(* Logix 5000 project; controller PBS_Perfusion vendor 1 type 14 code 217 rev 32.14; software revision 32.03; part 14 of 27 *)
(* tags used below, declared in another part *)
   Inp_OnFdbk : BOOL;   // Input Signal: ON feedback from device
   Inp_OffFdbk : BOOL;   // Input Signal: OFF feedback from device
   Inp_PermOK : BOOL;   // 1=ON Permissives OK, device can turn ON
   Inp_NBPermOK : BOOL;   // 1=Non-Bypassable ON Permissives OK, device can turn ON
   Inp_IntlkOK : BOOL;   // 1=Interlocks OK, device can turn ON and stay ON
   Inp_NBIntlkOK : BOOL;   // 1=Non-Bypassable Interlocks OK, device can turn ON and stay ON
   Inp_IntlkAvail : BOOL;   // 1 = Interlock Availibility OK
   Inp_IOFault : BOOL;   // Input Communication Status 0=OK, 1=fail
   Inp_Sim : BOOL;   // 1=Simulate working device; 0=Turn ON/OFF actual device
   Inp_OvrdCmd : DINT;   // Ovrd Device Command 0=None, 1=Off, 2=On, 3=Pulse Off, 4=Pulse On, 5=Pulse Cont
   Inp_HornInh : BOOL;   // 1 = Inhibit audible alert, 0 = Alllow audible alert
   Inp_Reset : BOOL;   // 1=Reset Shed Latches and Cleared Alarms
   Cfg_HasPulse : BOOL;   // 1=Enable pulsing functions, 0=On/Off only
   Cfg_HasOnFdbk : BOOL;   // 1=Device provides an ON feedback signal
   Cfg_HasOffFdbk : BOOL;   // 1=Device provides an OFF feedback signal
   Cfg_UseOnFdbk : BOOL;   // 1=Device ON feedback should be used for failure checking
   Cfg_UseOffFdbk : BOOL;   // 1=Device OFF feedback should be used for failure checking
   Cfg_FdbkFail : BOOL;   // 1=Both feedbacks ON is invalid; 0=Both feedbacks OFF is invalid
   Cfg_HasMoreObj : BOOL;   // 1=Tells HMI an object with more info is available
   Cfg_HornOnChange : BOOL;   // 0 = Horn on energize only, 1 = Horn on any state change
   Cfg_OperOffPrio : BOOL;   // 1=OCmd_Off any time, 0=OCmd_Off only when Oper selected
   Cfg_ExtOffPrio : BOOL;   // 1=XCmd_Off any time, 0=XCmd_Off only when Oper selected
   Cfg_OCmdResets : BOOL;   // 1=New device OCmd resets shed latches and cleared alarms, 0=OCmdReset req'd.
   Cfg_XCmdResets : BOOL;   // 1=New device XCmd resets shed latches and cleared alarms, 0=XCmdReset req'd.
   Cfg_OvrdPermIntlk : BOOL;   // 1=Override ignores Bypassable Perm/ Intlk; 0=always use Perm/Intlk
   Cfg_ShedOnFail : BOOL;   // 1=Go to State 0 and Alarm on Fail to reach position; 0=Alarm only on Fail
   Cfg_ShedOnIOFault : BOOL;   // 1=Go to State 0 and Alarm on I/O Fault; 0=Alarm only on I/O Fault
   Cfg_StartHornT : REAL;   // Time to sound audible on commanded start (sec) (0=disabled)
   Cfg_SimFdbkT : REAL;   // Delay to echo back of ON/OFF status when in Simulation (sec)
   Cfg_OnDelayT : REAL;   // Delay before initially turning output ON (sec)
   Cfg_OffDelayT : REAL;   // Delay before initially turning output OFF (sec)
   Cfg_OnPulseT : REAL;   // Output ON time for Pulse ON or Pulse Continuous
   Cfg_OffPulseT : REAL;   // Output OFF time for Pulse OFF or Pulse Continuous
   Cfg_OnFailT : REAL;   // Time after Output ON to get ON Feedback before Fault (sec)
   Cfg_OffFailT : REAL;   // Time after Output OFF to get OFF Feedback before Fault (sec)
   PSet_Owner : DINT;   // Program Owner Request ID (non-zero) or Release (zero)
   PCmd_On : BOOL;   // Program Command to turn device ON
   PCmd_Off : BOOL;   // Program Command to turn device OFF
   PCmd_OnPulse : BOOL;   // Program Command to pulse device (which is OFF) ON once
   PCmd_OffPulse : BOOL;   // Program Command to pulse device (which is ON) OFF once
   PCmd_ContPulse : BOOL;   // Program Command to pulse device continuously (blink)
   PCmd_Reset : BOOL;   // Program Command to ResetShed Latches and Cleared Alarms
   PCmd_OnFailAck : ALIAS FOR OnFail.PCmd_Ack;   // Program Command to Acknowledge Fail to Turn ON Alarm
   PCmd_OffFailAck : ALIAS FOR OffFail.PCmd_Ack;   // Program Command to Acknowledge Fail to Turn OFF Alarm
   PCmd_IntlkTripAck : ALIAS FOR IntlkTrip.PCmd_Ack;   // Program Command to Acknowledge Interlock Trip Alarm
   PCmd_IOFaultAck : ALIAS FOR IOFault.PCmd_Ack;   // Program Command to Acknowledge I/O Fault Alarm
   XCmd_On : BOOL;   // External Command to turn device ON
   XCmd_Off : BOOL;   // External Command to turn device OFF
   XCmd_OnPulse : BOOL;   // External Command to pulse device (which is OFF) ON once
   XCmd_OffPulse : BOOL;   // External Command to pulse device (which is ON) OFF once
   XCmd_ContPulse : BOOL;   // External Command to pulse device continuously (blink)
   XCmd_Reset : BOOL;   // Ext Cmd to clear shed latches and cleared alarms
   Out : BOOL;   // Primary Output 1=ON, 0=OFF
   Val_Fdbk : DINT;   // Device Feedback: 0=Transition, 1=Off, 2=On, 3=Invalid
   Val_Sts : DINT;   // Device Status 0=off 1=on 2=pulse off 3=pulse on 4=pulse cont. 5=turning off 6=turning on
   Val_Owner : DINT;   // Current Object Owner ID (0=not owned)
   Sts_FdbkOff : BOOL;   // 1=Device Feedback shows device in OFF state
   Sts_FdbkOn : BOOL;   // 1=Device Feedback shows device in ON state
   Sts_FdbkFail : BOOL;   // 1=Feedbacks are in an INVALID state (not ON, OFF or TRANSIT)
   Sts_Available : BOOL;   // 1=Device available for control by automation (Prog)
   Sts_Bypass : BOOL;   // 1=Bypassable Interlocks and Permissives are Bypassed
   Sts_BypActive : BOOL;   // 1=Interlock / Permissive Bypassing Active (Bypassed or Maintenance)
   Sts_NotRdy : BOOL;   // 1=Device Not Ready, see detail bits for reason
   Nrdy_CfgErr : BOOL;   // 1=Device Not Ready: Configuration Error
   Nrdy_Fail : BOOL;   // 1=Device Not Ready: Device Failure (Shed Requires Reset)
   Nrdy_Intlk : BOOL;   // 1=Device Not Ready: Interlock Not OK
   Nrdy_IOFault : BOOL;   // 1=Device Not Ready: I/O Fault (Shed Requires Reset)
   Nrdy_OoS : BOOL;   // 1=Device Not Ready: Device is Out of Service
   Nrdy_PrioOff : BOOL;   // 1=Device Not Ready: Oper/Ext Priority Off Comand Requires Reset
   Nrdy_Perm : BOOL;   // 1=Device Not Ready: Permissive Not OK
   Sts_MaintByp : BOOL;   // 1=Device has a Maintenance Bypass function active
   Err_Timer : BOOL;   // 1=Error in Config: Feeback Check timer preset (use 0 to 2147483)
   Err_Sim : BOOL;   // 1=Error in Config: Simulation timer preset (use 0 to 2147483)
   Sts_Hand : ALIAS FOR CmdSrc.Sts_Hand;
   Sts_OoS : ALIAS FOR CmdSrc.Sts_OoS;
   Sts_Maint : ALIAS FOR CmdSrc.Sts_Maint;
   Sts_Ovrd : ALIAS FOR CmdSrc.Sts_Ovrd;
   Sts_Ext : ALIAS FOR CmdSrc.Sts_Ext;
   Sts_Prog : ALIAS FOR CmdSrc.Sts_Prog;
   Sts_Oper : ALIAS FOR CmdSrc.Sts_Oper;
   Sts_OnFail : ALIAS FOR OnFail.Inp;   // 1=Device Failed to Turn ON
   Sts_OffFail : ALIAS FOR OffFail.Inp;   // 1=Device Failed to Turn OFF
   Sts_IntlkTrip : ALIAS FOR IntlkTrip.Inp;   // 1=Device turned OFF by an Interlock NOT OK (one-shot)
   Sts_IOFault : ALIAS FOR IOFault.Inp;   // I/O Comm Fault Status (0=OK, 1=Bad)
   P_DOut : BOOL;   // Unique Parameter Name for auto - discovery
   Wrk_OffT : TIMER;   // Off Feedback Check Timer
   Wrk_OnT : TIMER;   // On Feedback Check Timer
   Wrk_SimOffT : TIMER;   // Simulation Delay until OFF
   Wrk_SimOnT : TIMER;   // Simulation Delay until ON
   Wrk_OnFdbk : BOOL;   // ON Feedback based on Command Source, simulation, etc. 1=confirmed ON
   Wrk_Bypass : BOOL;   // Internal Bypassable Permissives and Interlocks are Bypassed flag
   CmdSrc : P_CmdSrc;   // Control / Command Source Selection
   IOFault : P_Alarm;   // I/O Fault Alarm
   IntlkTrip : P_Alarm;   // Interlock Trip Alarm
   OffFail : P_Alarm;   // Device Failed to Turn OFF Alarm
   OnFail : P_Alarm;   // Device Failed to Turn ON Alarm
   Cfg_Tag : STRING_20;   // Tagname for display on HMI
   Cfg_Label : STRING_20;   // Label for graphic symbol displayed on HMI
   Cfg_Desc : STRING_40;   // Description for display on HMI
   Wrk_OffFdbk : BOOL;   // OFF Feedback based on Command Source, simulation, etc. 1=confirmed OFF
   Wrk_OnPulseT : TIMER;   // Output ON Pulse Timer
   Wrk_OffPulseT : TIMER;   // Output OFF Pulse Timer
   Wrk_OffDelayT : TIMER;   // Dealy before turning output OFF (Timer)
   Wrk_OnDelayT : TIMER;   // Delay before turning output ON (Timer)
   Wrk_PermOK : BOOL;   // 1=Permissives are all OK to energize
   Wrk_Cmd : DINT;   // Device Command: 0= None, bit .0=Off, bit .1=On, bit .2=Pulse Off, bit .3=Pulse On, bit .4=Pulse Cont.
   Cfg_1StText : STRING_8;   // Text to display in PV=1 State
   Cfg_0StText : STRING_8;   // Text to display in PV=0 State
   HMI_Type : STRING_16;   // Type identifier for HMI navigation
   HMI_Lib : STRING_12;   // Display Library for Faceplate call-up
   Wrk_NotRdy : BOOL;   // Device Not Ready conditions excluding shed latches
   Wrk_NoLongerSim : BOOL;   // Switched from Simulated to Real Device this scan
   Cfg_Area : STRING_Area;   // Process Area for security
   OCmd_ResetAckAll : BOOL;   // Operator Command to Reset all Alarms and latched Shed conditions
   OCmd_Reset : BOOL;   // Operator Command to Reset all Alarms requiring Reset
   OCmd_ContPulse : BOOL;   // Operator Command to pulse device continuously (blink)
   OCmd_OffPulse : BOOL;   // Operator Command to pulse device (which is ON) OFF once
   OCmd_OnPulse : BOOL;   // Operator Command to pulse device (which is OFF) ON once
   OCmd_Off : BOOL;   // Operator Command to turn device OFF
   OCmd_On : BOOL;   // Operator Command to turn device ON
   MCmd_Check : BOOL;   // Maintenance Command to Check (not bypass) all Interlocks and Permissives
   MCmd_Bypass : BOOL;   // Maintenance Command to Bypass all Bypassable Interlocks and Permissives
   MRdy_Check : BOOL;   // 1=Ready for MCmd_Check (enables HMI button)
   MRdy_Bypass : BOOL;   // 1=Ready for MCmd_Bypass (enables HMI button)
   Wrk_State : DINT;   // Internal value of state machine current state
   Wrk_StartHornT : TIMER;   // Timer for audible alert or start
   Wrk_StartHorn : BOOL;   // 1=Sound audible prior to commanded energize/ state change
   ONS : DINT[3];
   REAL : DINT;
(* P_DOut, continued *)

ROUTINE Logic   (* ladder *)
// Control Discrete Output, monitoring Feedbacks
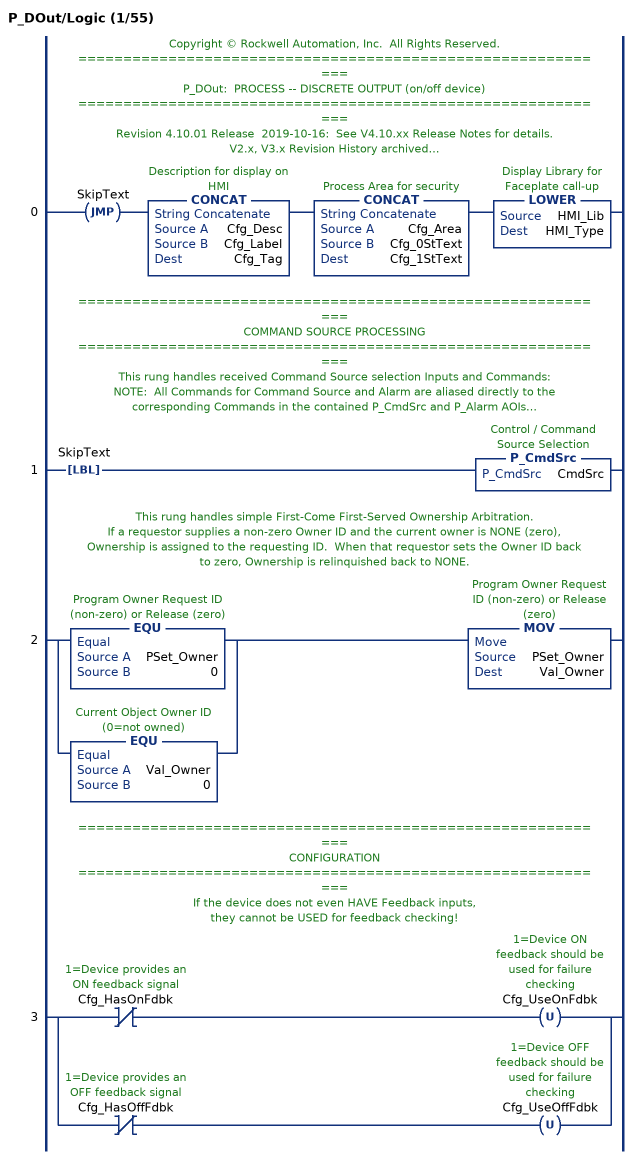
   // Copyright © Rockwell Automation, Inc.  All Rights Reserved.
   // ============================================================
   // P_DOut:  PROCESS -- DISCRETE OUTPUT (on/off device)
   // ============================================================
   // Revision 4.10.01 Release  2019-10-16:  See V4.10.xx Release Notes for details.
   // V2.x, V3.x Revision History archived.
   // V4.00.00  2018-07-02:  Changed "Mode" to "Command Source". Changed Inf_
   // items to HMI_, and added Cfg_Area for security. Added unacked alarm count.
   // Deleted Cfg_PCmdClear; all Program Commands are now self-clearing.
   // Added option: Cfg_HasPulse. Aligned ready bit naming with command bit names.
   // Changed delay / time configuration items to REAL seconds.
   // V4.00.02  2018-10-30:  Fixed feedback determination for simulation or no feedback.
   // V4.10.00  2019-10-16:  Added audible alert on commanded energize/state change.
   // Added Horn Status, Horn Inhibit. Changed availability to use input availability
   // from interlocks. Updated to P_CmdSrc V4.10.00. Added Cfg_HasMoreObj.
   // V4.10.01  2019-10-11:  Corrected operation of state machine with alert horn.
   // ============================================================
   // This Instruction controls (and optionally monitors feedback for)
   // a single Discrete Output and provides:
   // *  Operator and Program Commands to:
   //     -  turn the output ON
   //     -  turn the output OFF
   //     -  if the output is OFF, pulse it ON for a configured time
   //     -  if the output is ON, pulse it OFF for a configured time, or
   //     -  pulse the output continuously at the configured ON
   //         and OFF times (e.g., for blinking a lamp)
   // *  User-configurable ON delay and OFF delay before first output change
   // *  User-configurable text labels for the ON and OFF states
   // *  Optional monitoring of ON and OFF state confirmation feedbacks
   // *  Detection of Failure to turn ON or OFF (when feedbacks are used)
   // *  Monitoring of Permissive conditions to allow energizing output
   // *  Monitoring of Interlock conditions to de-energize output
   // *  Optional return to previous state upon return from Hand,
   //       Override, or Interlock
   // *  Simulation, providing feedback of a working device while
   //       disabling output (keeping de-energized)
   // *  Monitoring of I/O communication faults
   // *  Alarms for Fail to Turn ON, Fail to turn OFF (if feedbacks are
   //       used), Interlock Trip, I/O Fault
   // *  "Available" status for use by automation logic to know whether
   //       output can be controlled by other objects.
   // Command Sources are arbitrated by a P_CmdSrc Add-On Instruction instance.
   // Command Sources: Operator, External, Program, External, Override, Maintenance,
   // Out of Service, Hand.  Alarms are provided by P_Alarm Add-On Instruction instances.
   // ============================================================
   // SHOW LOCAL STRINGS
   // ============================================================
   // The STRINGs containing the text associated with each instance of this
   // instruction cannot be Input or Output Parameters, because STRINGs are not
   //  'atomic' types. (Inputs and Outputs must be SINT, INT, DINT, REAL, or BOOL.)
   // In order to make it easier to find and configure these STRINGs, this rung
   // was added.  THE JMP (and the LBL on the following rung)
   // MUST NOT BE REMOVED!!!
   // To view the STRINGs, go to the instruction instance (in LD or FBD), RIGHT-click
   // to bring up the context menu and select "Open Instruction Logic".
   // This rung will appear with the STRING values for the selected instance.
   // You may double-click the STRING values here to modify them as well.
   // #####  V4.00.00  2018-07-02:  Added string for Cfg_Area, renamed Inf_* to HMI_*.  #####
   0: JMP(SkipText)CONCAT(Cfg_Desc,Cfg_Label,Cfg_Tag)CONCAT(Cfg_Area,Cfg_0StText,Cfg_1StText)LOWER(HMI_Lib,HMI_Type);
   // ============================================================
   // COMMAND SOURCE PROCESSING
   // ============================================================
   // This rung handles received Command Source selection Inputs and Commands:
   // NOTE:  All Commands for Command Source and Alarm are aliased directly to the
   // corresponding Commands in the contained P_CmdSrc and P_Alarm AOIs.
   // #####  V4.00.00  2018-07-02:  Changed P_Mode to P_CmdSrc.  #####
   1: LBL(SkipText)P_CmdSrc(CmdSrc);
   // This rung handles simple First-Come First-Served Ownership Arbitration.
   // If a requestor supplies a non-zero Owner ID and the current owner is NONE (zero),
   // Ownership is assigned to the requesting ID.  When that requestor sets the Owner ID back
   // to zero, Ownership is relinquished back to NONE.
   2: [EQU(PSet_Owner,0) ,EQU(Val_Owner,0) ]MOV(PSet_Owner,Val_Owner);
   // ============================================================
   // CONFIGURATION
   // ============================================================
   // If the device does not even HAVE Feedback inputs,
   // they cannot be USED for feedback checking!
   3: [XIO(Cfg_HasOnFdbk) OTU(Cfg_UseOnFdbk) ,XIO(Cfg_HasOffFdbk) OTU(Cfg_UseOffFdbk) ];
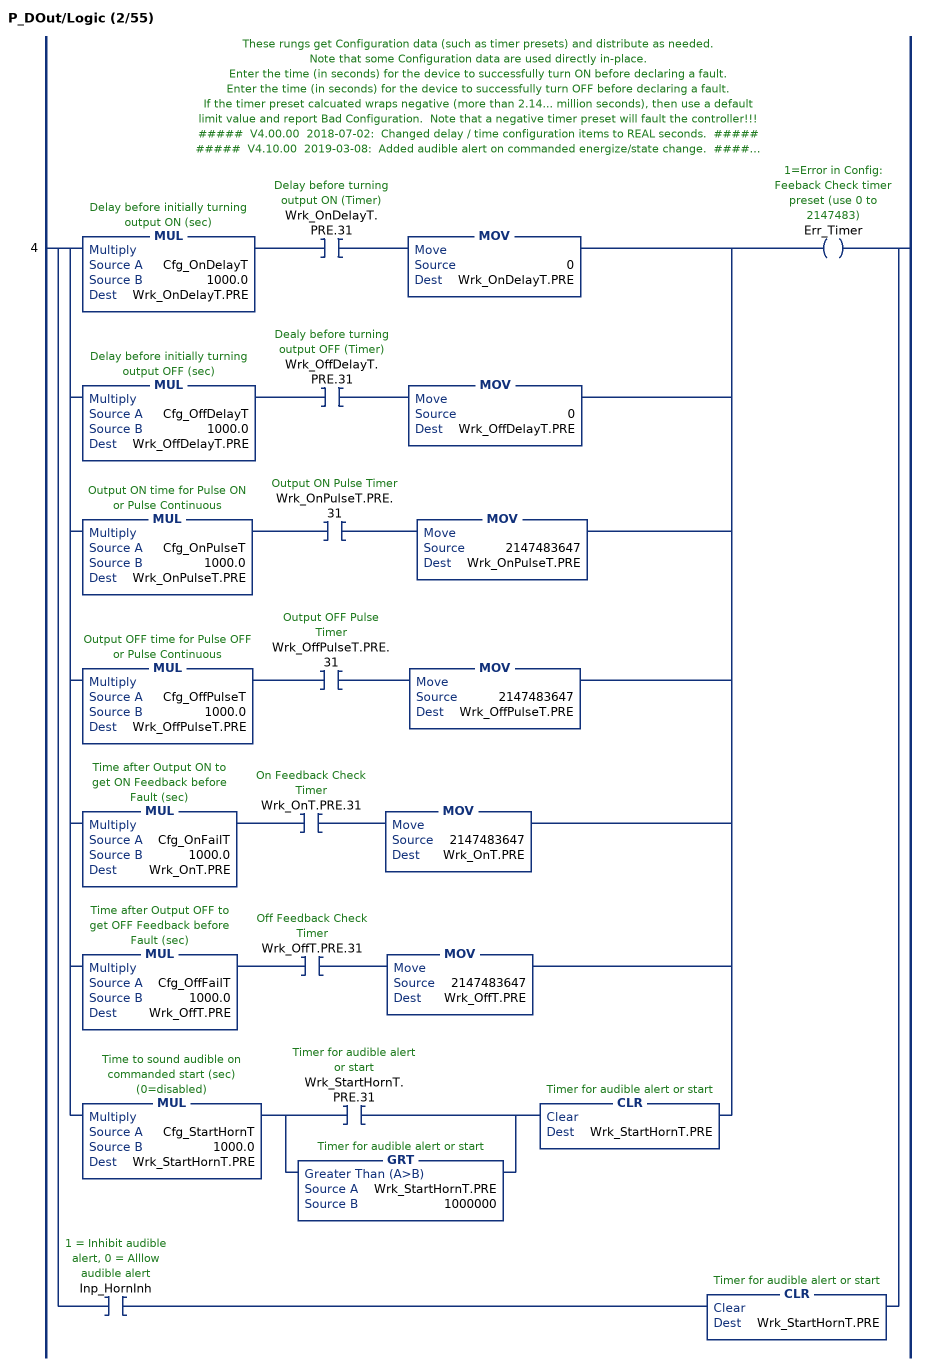
   // These rungs get Configuration data (such as timer presets) and distribute as needed.
   // Note that some Configuration data are used directly in-place.
   // Enter the time (in seconds) for the device to successfully turn ON before declaring a fault.
   // Enter the time (in seconds) for the device to successfully turn OFF before declaring a fault.
   // If the timer preset calcuated wraps negative (more than 2.14... million seconds), then use a default
   // limit value and report Bad Configuration.  Note that a negative timer preset will fault the controller!!!
   // #####  V4.00.00  2018-07-02:  Changed delay / time configuration items to REAL seconds.  #####
   // #####  V4.10.00  2019-03-08:  Added audible alert on commanded energize/state change.  #####
   // #####  Added Inp_HornInh to disable Horn operation.  #####
   4: [[MUL(Cfg_OnDelayT,1000.0,Wrk_OnDelayT.PRE) XIC(Wrk_OnDelayT.PRE.31) MOV(0,Wrk_OnDelayT.PRE) ,MUL(Cfg_OffDelayT,1000.0,Wrk_OffDelayT.PRE) XIC(Wrk_OffDelayT.PRE.31) MOV(0,Wrk_OffDelayT.PRE) ,MUL(Cfg_OnPulseT,1000.0,Wrk_OnPulseT.PRE) XIC(Wrk_OnPulseT.PRE.31) MOV(2147483647,Wrk_OnPulseT.PRE) ,MUL(Cfg_OffPulseT,1000.0,Wrk_OffPulseT.PRE) XIC(Wrk_OffPulseT.PRE.31) MOV(2147483647,Wrk_OffPulseT.PRE) ,MUL(Cfg_OnFailT,1000.0,Wrk_OnT.PRE) XIC(Wrk_OnT.PRE.31) MOV(2147483647,Wrk_OnT.PRE) ,MUL(Cfg_OffFailT,1000.0,Wrk_OffT.PRE) XIC(Wrk_OffT.PRE.31) MOV(2147483647,Wrk_OffT.PRE) ,MUL(Cfg_StartHornT,1000.0,Wrk_StartHornT.PRE) [XIC(Wrk_StartHornT.PRE.31) ,GRT(Wrk_StartHornT.PRE,1000000) ] CLR(Wrk_StartHornT.PRE) ] OTE(Err_Timer) ,XIC(Inp_HornInh) CLR(Wrk_StartHornT.PRE) ];
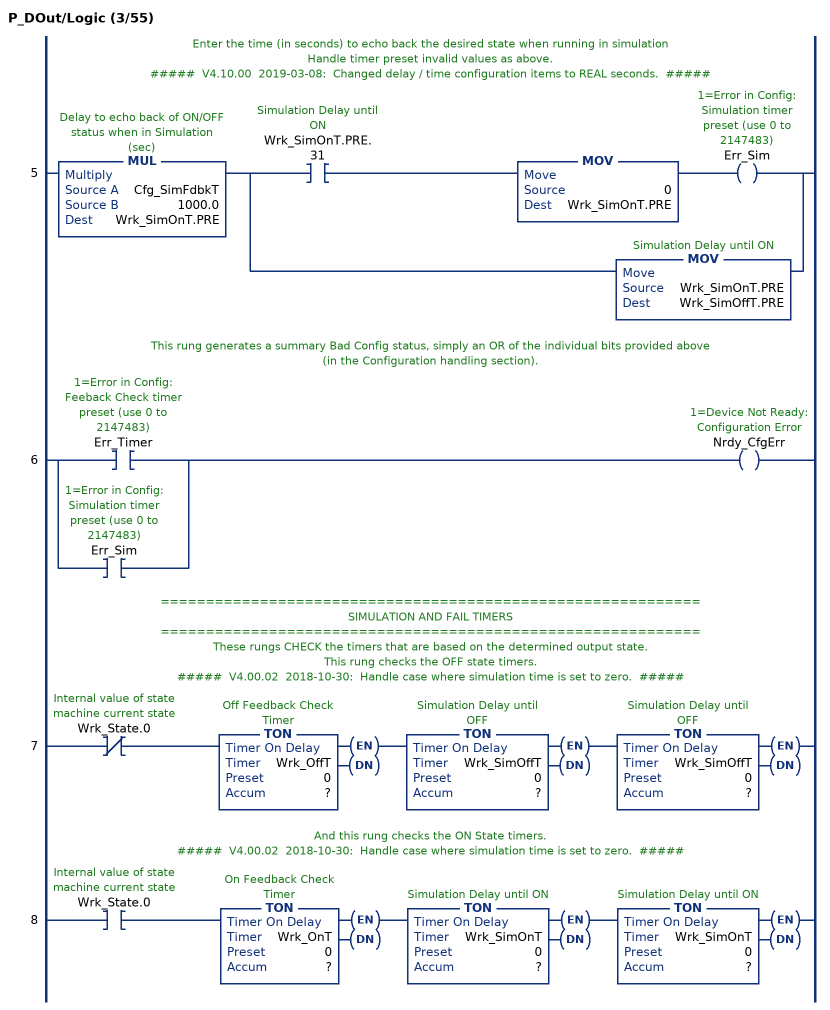
   // Enter the time (in seconds) to echo back the desired state when running in simulation
   // Handle timer preset invalid values as above.
   // #####  V4.10.00  2019-03-08:  Changed delay / time configuration items to REAL seconds.  #####
   5: MUL(Cfg_SimFdbkT,1000.0,Wrk_SimOnT.PRE)[XIC(Wrk_SimOnT.PRE.31) MOV(0,Wrk_SimOnT.PRE) OTE(Err_Sim) ,MOV(Wrk_SimOnT.PRE,Wrk_SimOffT.PRE) ];
   // This rung generates a summary Bad Config status, simply an OR of the individual bits provided above
   // (in the Configuration handling section).
   6: [XIC(Err_Timer) ,XIC(Err_Sim) ]OTE(Nrdy_CfgErr);
   // ============================================================
   // SIMULATION AND FAIL TIMERS
   // ============================================================
   // These rungs CHECK the timers that are based on the determined output state.
   // This rung checks the OFF state timers.
   // #####  V4.00.02  2018-10-30:  Handle case where simulation time is set to zero.  #####
   7: XIO(Wrk_State.0)TON(Wrk_OffT,?,?)TON(Wrk_SimOffT,?,?)TON(Wrk_SimOffT,?,?);
   // And this rung checks the ON State timers.
   // #####  V4.00.02  2018-10-30:  Handle case where simulation time is set to zero.  #####
   8: XIC(Wrk_State.0)TON(Wrk_OnT,?,?)TON(Wrk_SimOnT,?,?)TON(Wrk_SimOnT,?,?);
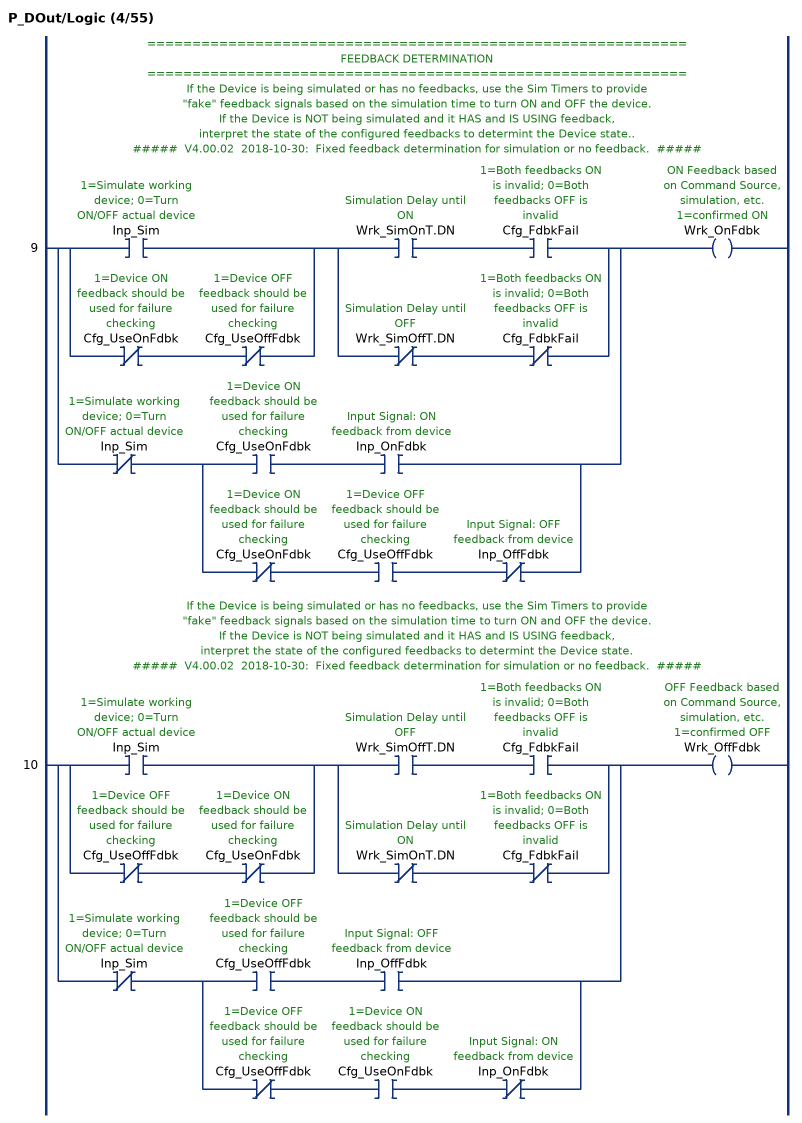
   // ============================================================
   // FEEDBACK DETERMINATION
   // ============================================================
   // If the Device is being simulated or has no feedbacks, use the Sim Timers to provide
   // "fake" feedback signals based on the simulation time to turn ON and OFF the device.
   // If the Device is NOT being simulated and it HAS and IS USING feedback,
   // interpret the state of the configured feedbacks to determint the Device state..
   // #####  V4.00.02  2018-10-30:  Fixed feedback determination for simulation or no feedback.  #####
   9: [[XIC(Inp_Sim) ,XIO(Cfg_UseOnFdbk) XIO(Cfg_UseOffFdbk) ] [XIC(Wrk_SimOnT.DN) XIC(Cfg_FdbkFail) ,XIO(Wrk_SimOffT.DN) XIO(Cfg_FdbkFail) ] ,XIO(Inp_Sim) [XIC(Cfg_UseOnFdbk) XIC(Inp_OnFdbk) ,XIO(Cfg_UseOnFdbk) XIC(Cfg_UseOffFdbk) XIO(Inp_OffFdbk) ] ]OTE(Wrk_OnFdbk);
   // If the Device is being simulated or has no feedbacks, use the Sim Timers to provide
   // "fake" feedback signals based on the simulation time to turn ON and OFF the device.
   // If the Device is NOT being simulated and it HAS and IS USING feedback,
   // interpret the state of the configured feedbacks to determint the Device state.
   // #####  V4.00.02  2018-10-30:  Fixed feedback determination for simulation or no feedback.  #####
   10: [[XIC(Inp_Sim) ,XIO(Cfg_UseOffFdbk) XIO(Cfg_UseOnFdbk) ] [XIC(Wrk_SimOffT.DN) XIC(Cfg_FdbkFail) ,XIO(Wrk_SimOnT.DN) XIO(Cfg_FdbkFail) ] ,XIO(Inp_Sim) [XIC(Cfg_UseOffFdbk) XIC(Inp_OffFdbk) ,XIO(Cfg_UseOffFdbk) XIC(Cfg_UseOnFdbk) XIO(Inp_OnFdbk) ] ]OTE(Wrk_OffFdbk);
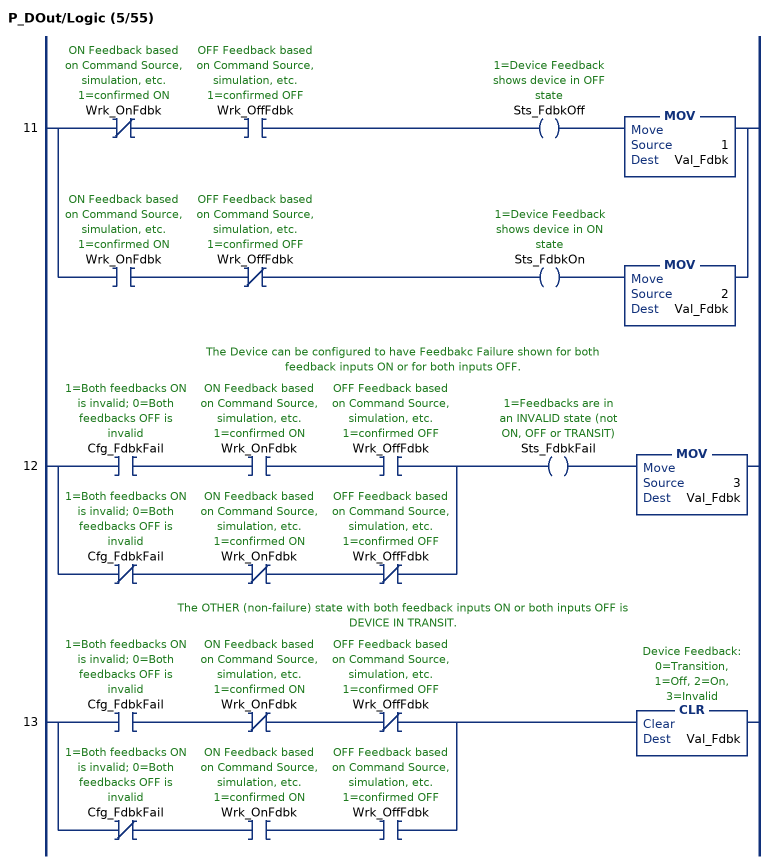
   11: [XIO(Wrk_OnFdbk) XIC(Wrk_OffFdbk) OTE(Sts_FdbkOff) MOV(1,Val_Fdbk) ,XIC(Wrk_OnFdbk) XIO(Wrk_OffFdbk) OTE(Sts_FdbkOn) MOV(2,Val_Fdbk) ];
   // The Device can be configured to have Feedbakc Failure shown for both
   // feedback inputs ON or for both inputs OFF.
   12: [XIC(Cfg_FdbkFail) XIC(Wrk_OnFdbk) XIC(Wrk_OffFdbk) ,XIO(Cfg_FdbkFail) XIO(Wrk_OnFdbk) XIO(Wrk_OffFdbk) ]OTE(Sts_FdbkFail)MOV(3,Val_Fdbk);
   // The OTHER (non-failure) state with both feedback inputs ON or both inputs OFF is
   // DEVICE IN TRANSIT.
   13: [XIC(Cfg_FdbkFail) XIO(Wrk_OnFdbk) XIO(Wrk_OffFdbk) ,XIO(Cfg_FdbkFail) XIC(Wrk_OnFdbk) XIC(Wrk_OffFdbk) ]CLR(Val_Fdbk);
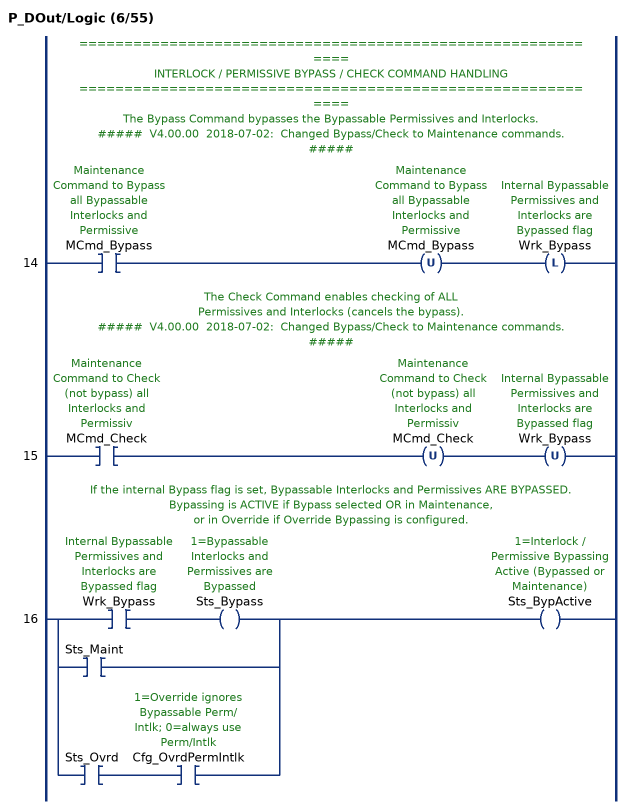
   // ============================================================
   // INTERLOCK / PERMISSIVE BYPASS / CHECK COMMAND HANDLING
   // ============================================================
   // The Bypass Command bypasses the Bypassable Permissives and Interlocks.
   // #####  V4.00.00  2018-07-02:  Changed Bypass/Check to Maintenance commands.  #####
   14: XIC(MCmd_Bypass)OTU(MCmd_Bypass)OTL(Wrk_Bypass);
   // The Check Command enables checking of ALL
   // Permissives and Interlocks (cancels the bypass).
   // #####  V4.00.00  2018-07-02:  Changed Bypass/Check to Maintenance commands.  #####
   15: XIC(MCmd_Check)OTU(MCmd_Check)OTU(Wrk_Bypass);
   // If the internal Bypass flag is set, Bypassable Interlocks and Permissives ARE BYPASSED.
   // Bypassing is ACTIVE if Bypass selected OR in Maintenance,
   // or in Override if Override Bypassing is configured.
   16: [XIC(Wrk_Bypass) OTE(Sts_Bypass) ,XIC(Sts_Maint) ,XIC(Sts_Ovrd) XIC(Cfg_OvrdPermIntlk) ]OTE(Sts_BypActive);
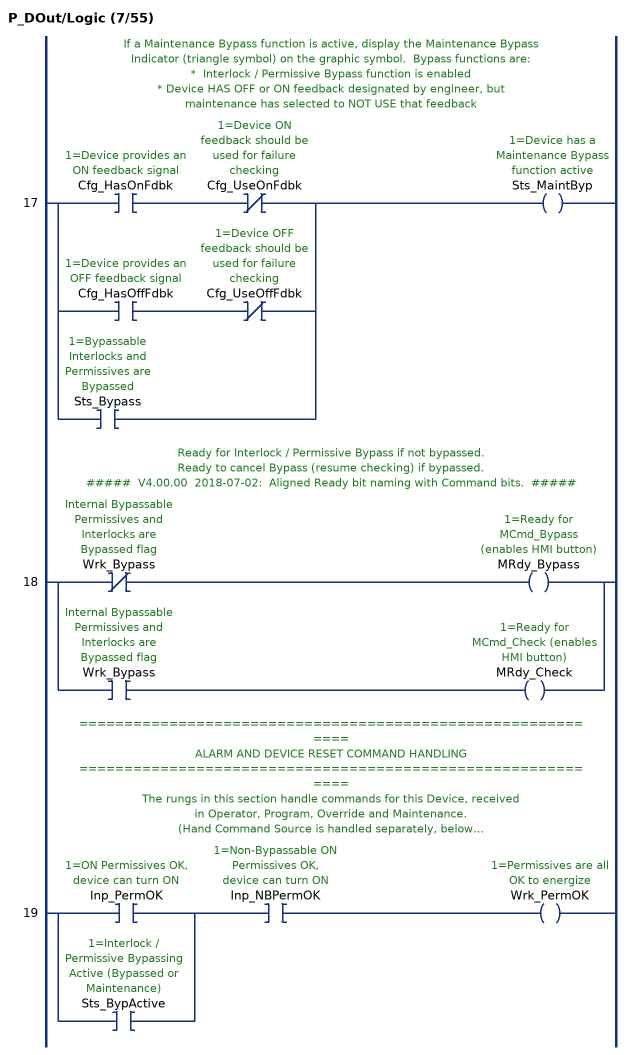
   // If a Maintenance Bypass function is active, display the Maintenance Bypass
   // Indicator (triangle symbol) on the graphic symbol.  Bypass functions are:
   // *  Interlock / Permissive Bypass function is enabled
   // * Device HAS OFF or ON feedback designated by engineer, but
   // maintenance has selected to NOT USE that feedback
   17: [XIC(Cfg_HasOnFdbk) XIO(Cfg_UseOnFdbk) ,XIC(Cfg_HasOffFdbk) XIO(Cfg_UseOffFdbk) ,XIC(Sts_Bypass) ]OTE(Sts_MaintByp);
   // Ready for Interlock / Permissive Bypass if not bypassed.
   // Ready to cancel Bypass (resume checking) if bypassed.
   // #####  V4.00.00  2018-07-02:  Aligned Ready bit naming with Command bits.  #####
   18: [XIO(Wrk_Bypass) OTE(MRdy_Bypass) ,XIC(Wrk_Bypass) OTE(MRdy_Check) ];
   // ============================================================
   // ALARM AND DEVICE RESET COMMAND HANDLING
   // ============================================================
   // The rungs in this section handle commands for this Device, received
   // in Operator, Program, Override and Maintenance.
   // (Hand Command Source is handled separately, below.
   // For any command which involves energizing the device (all commands
   // except OFF), permissives must be OK to energize.
   19: [XIC(Inp_PermOK) ,XIC(Sts_BypActive) ]XIC(Inp_NBPermOK)OTE(Wrk_PermOK);
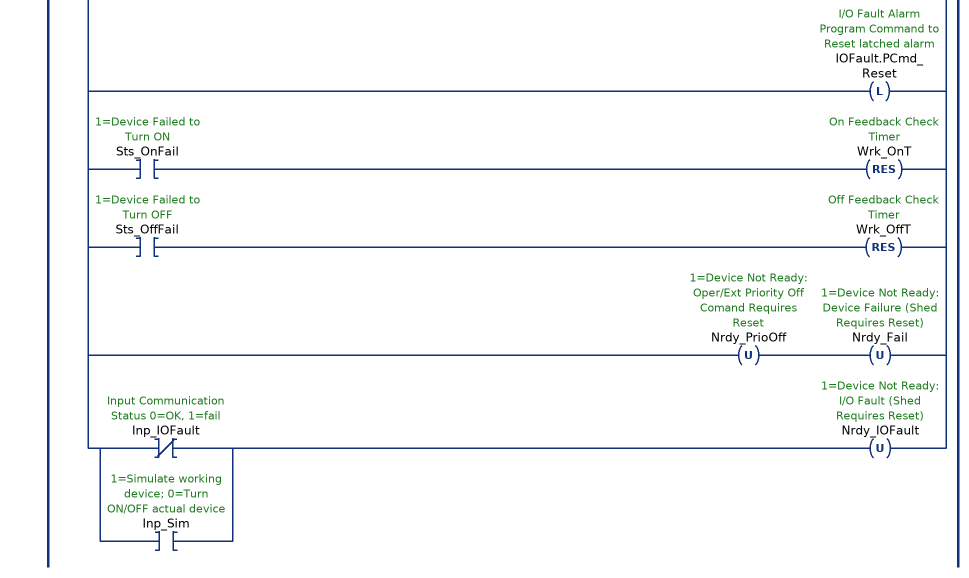
   // ============================================================
   // ALARM RESET COMMAND HANDLING
   // ============================================================
   // This rung handles the Alarm Reset Input and Commands
   // and the "Reset and Ack All" Operator Command.
   // This rung processes received Reset Commands from:
   // 1.  The Operator via HMI Operator Command, or
   // 2.  Higher-level strategies via Program Command
   // 3.  Pushbuttons or other block via Input
   // 4.  Resets initiated by other device Operator Commands (if configured to do so)
   // and forwards the Reset to ALL Alarms and latched Shed conditions.
   // #####  V4.00.00  2018-07-02:  Deleted Cfg_PCmdClear; all Program Commands are now self-clearing.  #####
   // #####  Added External Command Source and Commands.  #####
   20: [XIC(OCmd_Reset) OTU(OCmd_Reset) ,XIC(XCmd_Reset) OTU(XCmd_Reset) ,XIC(PCmd_Reset) OTU(PCmd_Reset) ,XIC(Inp_Reset) ,[XIC(OCmd_Off) ,[XIC(OCmd_On) ,XIC(Cfg_HasPulse) [XIC(OCmd_OffPulse) ,XIC(OCmd_OnPulse) ,XIC(OCmd_ContPulse) ] ] XIC(Wrk_PermOK) ] XIC(Cfg_OCmdResets) XIO(Nrdy_CfgErr) [XIC(Sts_Oper) ,XIC(Sts_Maint) ] ,[XIC(XCmd_Off) ,[XIC(XCmd_On) ,XIC(Cfg_HasPulse) [XIC(XCmd_OffPulse) ,XIC(XCmd_OnPulse) ,XIC(XCmd_ContPulse) ] ] XIC(Wrk_PermOK) ] XIC(Cfg_XCmdResets) XIO(Nrdy_CfgErr) XIC(Sts_Ext) ,XIC(OCmd_ResetAckAll) OTU(OCmd_ResetAckAll) [OTL(PCmd_OnFailAck) ,OTL(PCmd_OffFailAck) ,OTL(PCmd_IntlkTripAck) ,OTL(PCmd_IOFaultAck) ] ][OTL(OnFail.PCmd_Reset) ,OTL(OffFail.PCmd_Reset) ,OTL(IntlkTrip.PCmd_Reset) ,OTL(IOFault.PCmd_Reset) ,XIC(Sts_OnFail) RES(Wrk_OnT) ,XIC(Sts_OffFail) RES(Wrk_OffT) ,OTU(Nrdy_PrioOff) OTU(Nrdy_Fail) ,[XIO(Inp_IOFault) ,XIC(Inp_Sim) ] OTU(Nrdy_IOFault) ];
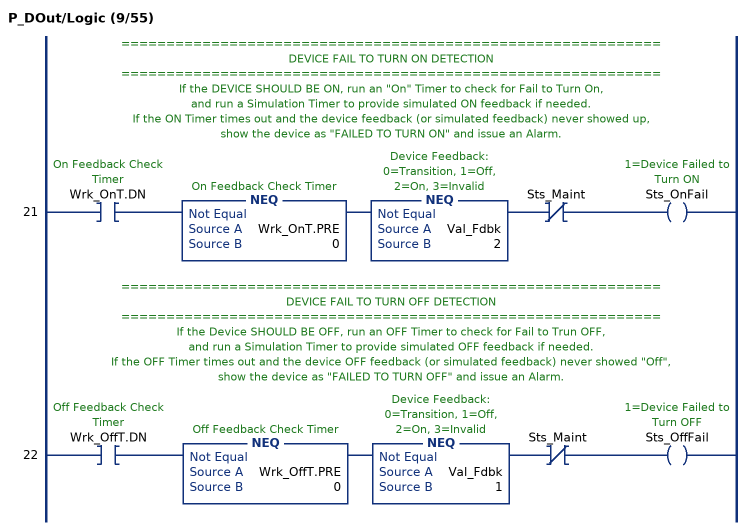
   // ============================================================
   // DEVICE FAIL TO TURN ON DETECTION
   // ============================================================
   // If the DEVICE SHOULD BE ON, run an "On" Timer to check for Fail to Turn On,
   // and run a Simulation Timer to provide simulated ON feedback if needed.
   // If the ON Timer times out and the device feedback (or simulated feedback) never showed up,
   // show the device as "FAILED TO TURN ON" and issue an Alarm.
   21: XIC(Wrk_OnT.DN)NEQ(Wrk_OnT.PRE,0)NEQ(Val_Fdbk,2)XIO(Sts_Maint)OTE(Sts_OnFail);
   // ============================================================
   // DEVICE FAIL TO TURN OFF DETECTION
   // ============================================================
   // If the Device SHOULD BE OFF, run an OFF Timer to check for Fail to Trun OFF,
   // and run a Simulation Timer to provide simulated OFF feedback if needed.
   // If the OFF Timer times out and the device OFF feedback (or simulated feedback) never showed "Off",
   // show the device as "FAILED TO TURN OFF" and issue an Alarm.
   22: XIC(Wrk_OffT.DN)NEQ(Wrk_OffT.PRE,0)NEQ(Val_Fdbk,1)XIO(Sts_Maint)OTE(Sts_OffFail);
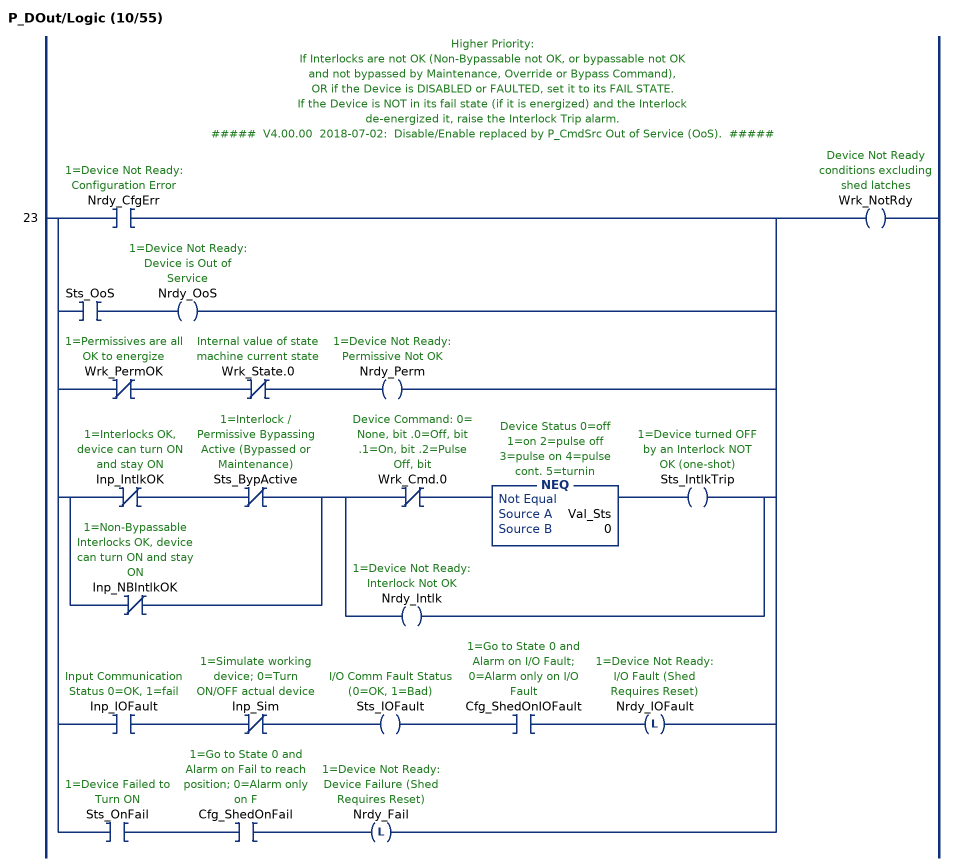
   // Higher Priority:
   // If Interlocks are not OK (Non-Bypassable not OK, or bypassable not OK
   // and not bypassed by Maintenance, Override or Bypass Command),
   // OR if the Device is DISABLED or FAULTED, set it to its FAIL STATE.
   // If the Device is NOT in its fail state (if it is energized) and the Interlock
   // de-energized it, raise the Interlock Trip alarm.
   // #####  V4.00.00  2018-07-02:  Disable/Enable replaced by P_CmdSrc Out of Service (OoS).  #####
   23: [XIC(Nrdy_CfgErr) ,XIC(Sts_OoS) OTE(Nrdy_OoS) ,XIO(Wrk_PermOK) XIO(Wrk_State.0) OTE(Nrdy_Perm) ,[XIO(Inp_IntlkOK) XIO(Sts_BypActive) ,XIO(Inp_NBIntlkOK) ] [XIO(Wrk_Cmd.0) NEQ(Val_Sts,0) OTE(Sts_IntlkTrip) ,OTE(Nrdy_Intlk) ] ,XIC(Inp_IOFault) XIO(Inp_Sim) OTE(Sts_IOFault) XIC(Cfg_ShedOnIOFault) OTL(Nrdy_IOFault) ,XIC(Sts_OnFail) XIC(Cfg_ShedOnFail) OTL(Nrdy_Fail) ]OTE(Wrk_NotRdy);
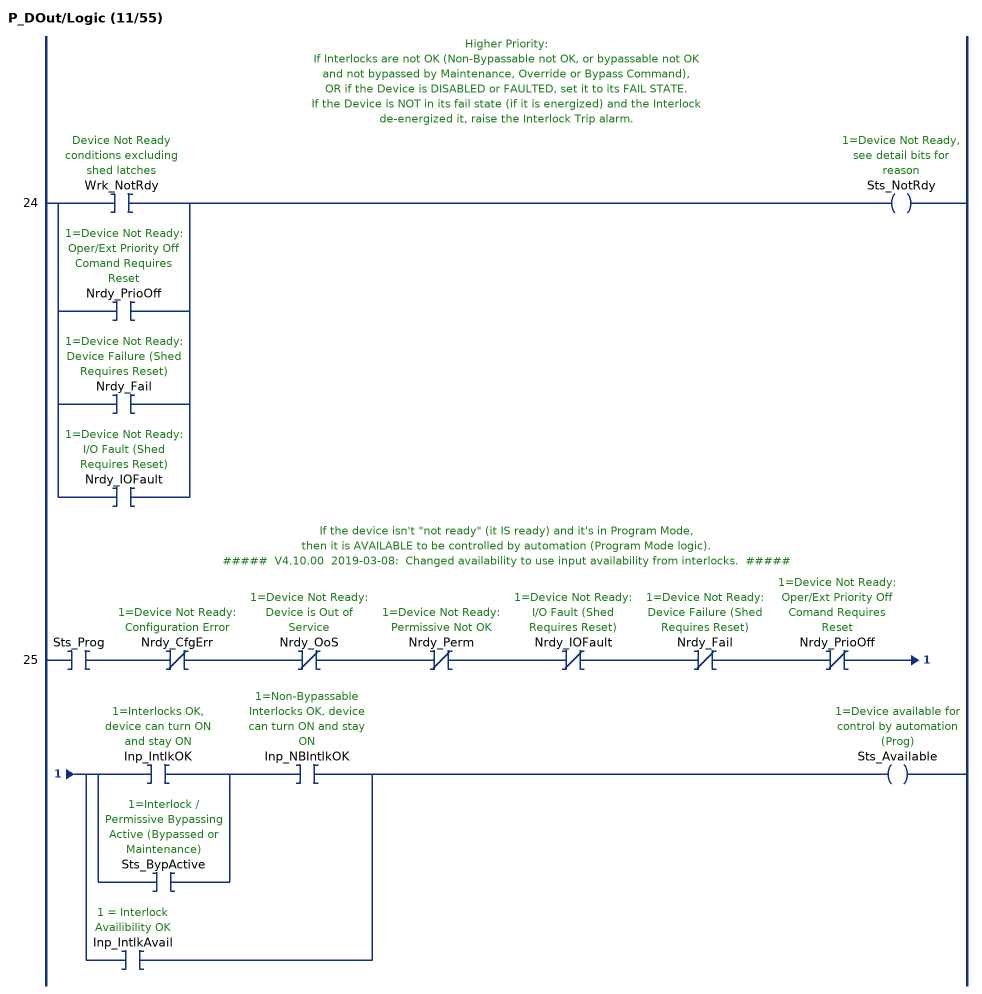
   // Higher Priority:
   // If Interlocks are not OK (Non-Bypassable not OK, or bypassable not OK
   // and not bypassed by Maintenance, Override or Bypass Command),
   // OR if the Device is DISABLED or FAULTED, set it to its FAIL STATE.
   // If the Device is NOT in its fail state (if it is energized) and the Interlock
   // de-energized it, raise the Interlock Trip alarm.
   24: [XIC(Wrk_NotRdy) ,XIC(Nrdy_PrioOff) ,XIC(Nrdy_Fail) ,XIC(Nrdy_IOFault) ]OTE(Sts_NotRdy);
   // If the device isn't "not ready" (it IS ready) and it's in Program Mode,
   // then it is AVAILABLE to be controlled by automation (Program Mode logic).
   // #####  V4.10.00  2019-03-08:  Changed availability to use input availability from interlocks.  #####
   25: XIC(Sts_Prog)XIO(Nrdy_CfgErr)XIO(Nrdy_OoS)XIO(Nrdy_Perm)XIO(Nrdy_IOFault)XIO(Nrdy_Fail)XIO(Nrdy_PrioOff)[[XIC(Inp_IntlkOK) ,XIC(Sts_BypActive) ] XIC(Inp_NBIntlkOK) ,XIC(Inp_IntlkAvail) ]OTE(Sts_Available);
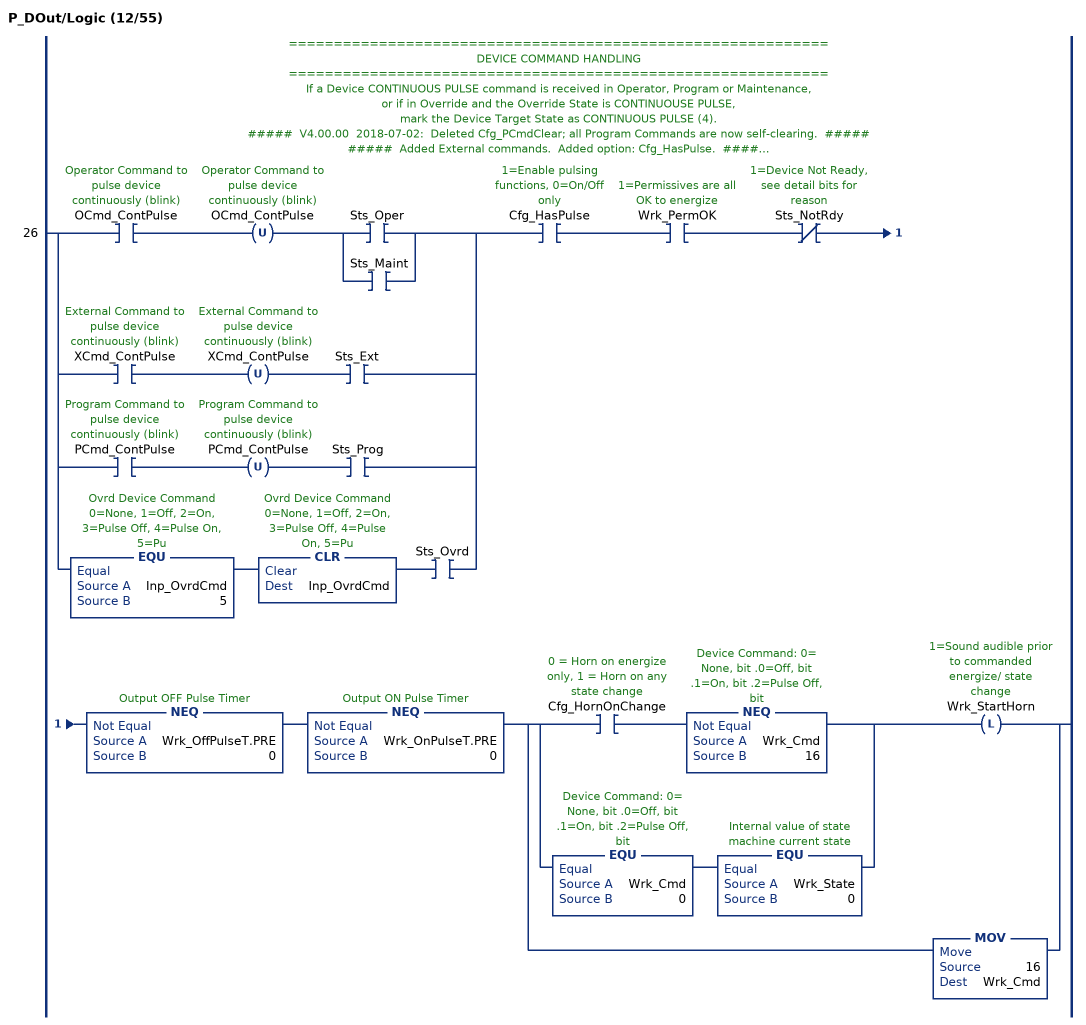
   // ============================================================
   // DEVICE COMMAND HANDLING
   // ============================================================
   // If a Device CONTINUOUS PULSE command is received in Operator, Program or Maintenance,
   // or if in Override and the Override State is CONTINUOUSE PULSE,
   // mark the Device Target State as CONTINUOUS PULSE (4).
   // #####  V4.00.00  2018-07-02:  Deleted Cfg_PCmdClear; all Program Commands are now self-clearing.  #####
   // #####  Added External commands.  Added option: Cfg_HasPulse.  #####
   // #####  V4.10.00  2019-03-08:  Added audible alert on commanded energize/state change.  #####
   // #####  V4.10.01  2019-10-16:  Corrected operation of state machine with alert horn.  #####
   26: [XIC(OCmd_ContPulse) OTU(OCmd_ContPulse) [XIC(Sts_Oper) ,XIC(Sts_Maint) ] ,XIC(XCmd_ContPulse) OTU(XCmd_ContPulse) XIC(Sts_Ext) ,XIC(PCmd_ContPulse) OTU(PCmd_ContPulse) XIC(Sts_Prog) ,EQU(Inp_OvrdCmd,5) CLR(Inp_OvrdCmd) XIC(Sts_Ovrd) ]XIC(Cfg_HasPulse)XIC(Wrk_PermOK)XIO(Sts_NotRdy)NEQ(Wrk_OffPulseT.PRE,0)NEQ(Wrk_OnPulseT.PRE,0)[[XIC(Cfg_HornOnChange) NEQ(Wrk_Cmd,16) ,EQU(Wrk_Cmd,0) EQU(Wrk_State,0) ] OTL(Wrk_StartHorn) ,MOV(16,Wrk_Cmd) ];
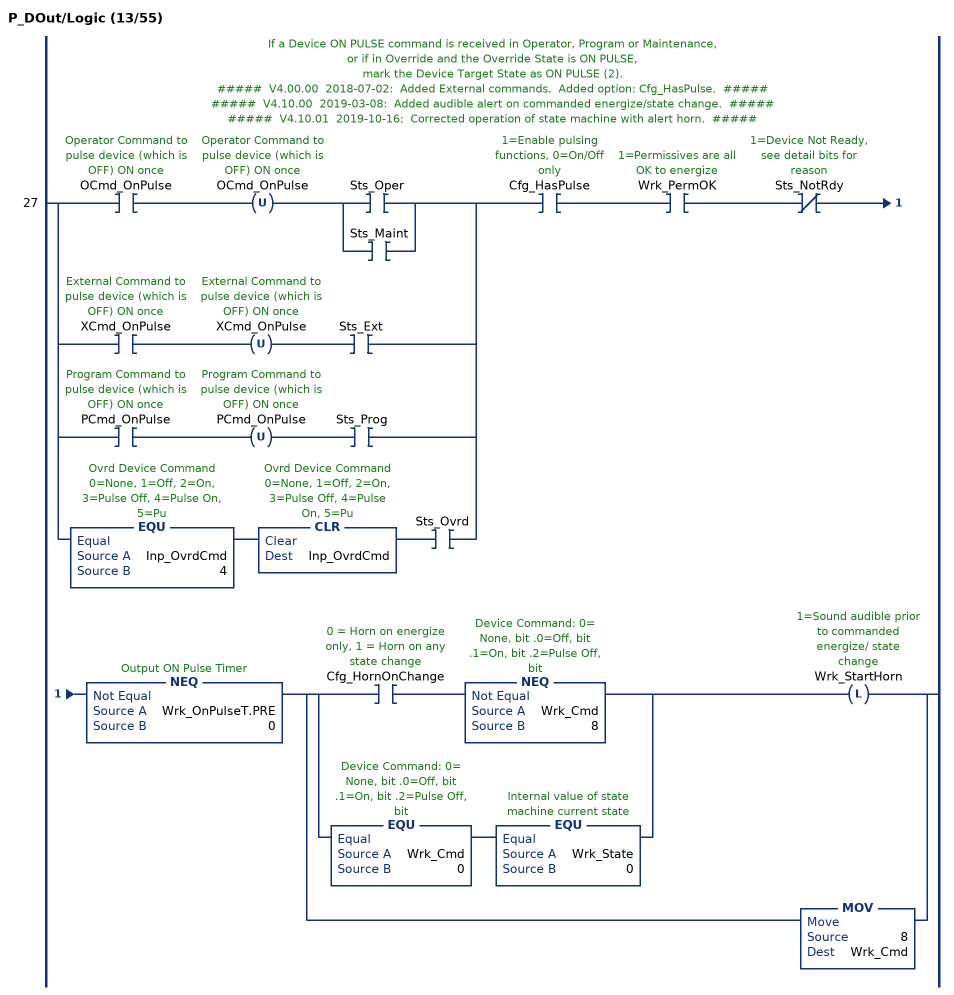
   // If a Device ON PULSE command is received in Operator, Program or Maintenance,
   // or if in Override and the Override State is ON PULSE,
   // mark the Device Target State as ON PULSE (2).
   // #####  V4.00.00  2018-07-02:  Added External commands.  Added option: Cfg_HasPulse.  #####
   // #####  V4.10.00  2019-03-08:  Added audible alert on commanded energize/state change.  #####
   // #####  V4.10.01  2019-10-16:  Corrected operation of state machine with alert horn.  #####
   27: [XIC(OCmd_OnPulse) OTU(OCmd_OnPulse) [XIC(Sts_Oper) ,XIC(Sts_Maint) ] ,XIC(XCmd_OnPulse) OTU(XCmd_OnPulse) XIC(Sts_Ext) ,XIC(PCmd_OnPulse) OTU(PCmd_OnPulse) XIC(Sts_Prog) ,EQU(Inp_OvrdCmd,4) CLR(Inp_OvrdCmd) XIC(Sts_Ovrd) ]XIC(Cfg_HasPulse)XIC(Wrk_PermOK)XIO(Sts_NotRdy)NEQ(Wrk_OnPulseT.PRE,0)[[XIC(Cfg_HornOnChange) NEQ(Wrk_Cmd,8) ,EQU(Wrk_Cmd,0) EQU(Wrk_State,0) ] OTL(Wrk_StartHorn) ,MOV(8,Wrk_Cmd) ];
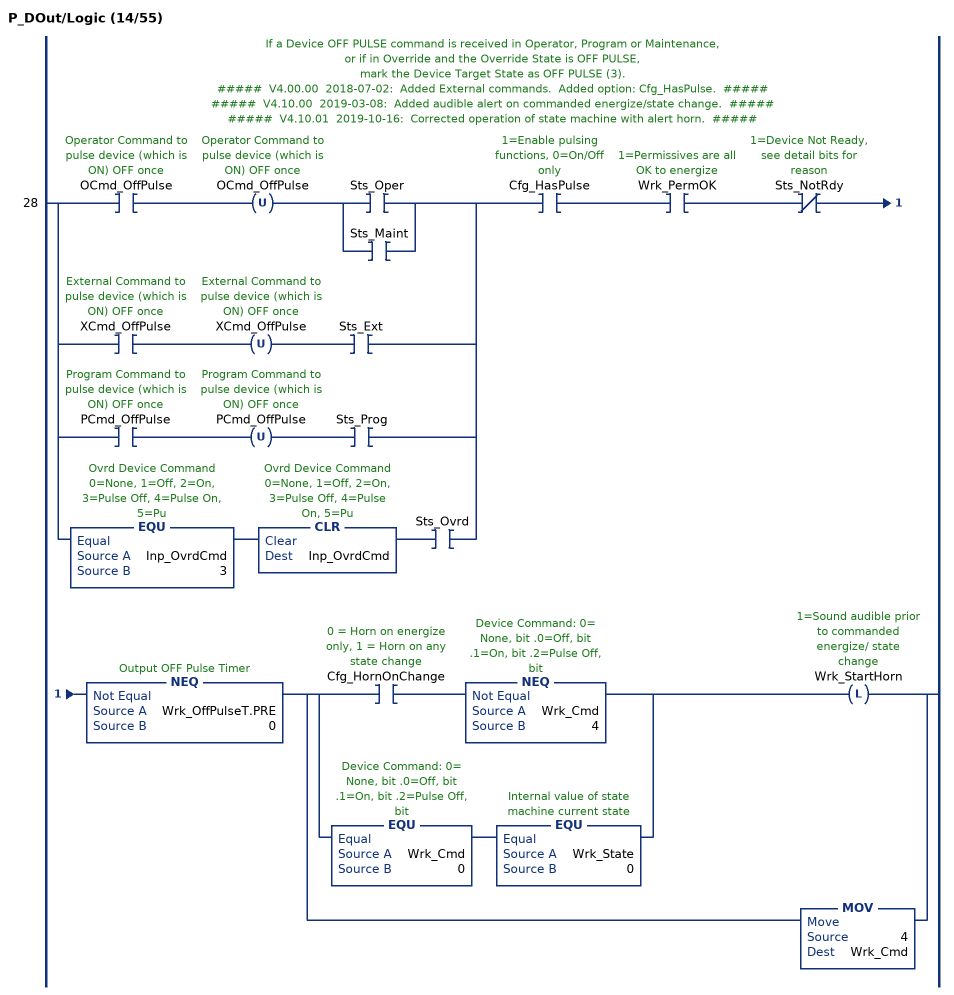
   // If a Device OFF PULSE command is received in Operator, Program or Maintenance,
   // or if in Override and the Override State is OFF PULSE,
   // mark the Device Target State as OFF PULSE (3).
   // #####  V4.00.00  2018-07-02:  Added External commands.  Added option: Cfg_HasPulse.  #####
   // #####  V4.10.00  2019-03-08:  Added audible alert on commanded energize/state change.  #####
   // #####  V4.10.01  2019-10-16:  Corrected operation of state machine with alert horn.  #####
   28: [XIC(OCmd_OffPulse) OTU(OCmd_OffPulse) [XIC(Sts_Oper) ,XIC(Sts_Maint) ] ,XIC(XCmd_OffPulse) OTU(XCmd_OffPulse) XIC(Sts_Ext) ,XIC(PCmd_OffPulse) OTU(PCmd_OffPulse) XIC(Sts_Prog) ,EQU(Inp_OvrdCmd,3) CLR(Inp_OvrdCmd) XIC(Sts_Ovrd) ]XIC(Cfg_HasPulse)XIC(Wrk_PermOK)XIO(Sts_NotRdy)NEQ(Wrk_OffPulseT.PRE,0)[[XIC(Cfg_HornOnChange) NEQ(Wrk_Cmd,4) ,EQU(Wrk_Cmd,0) EQU(Wrk_State,0) ] OTL(Wrk_StartHorn) ,MOV(4,Wrk_Cmd) ];
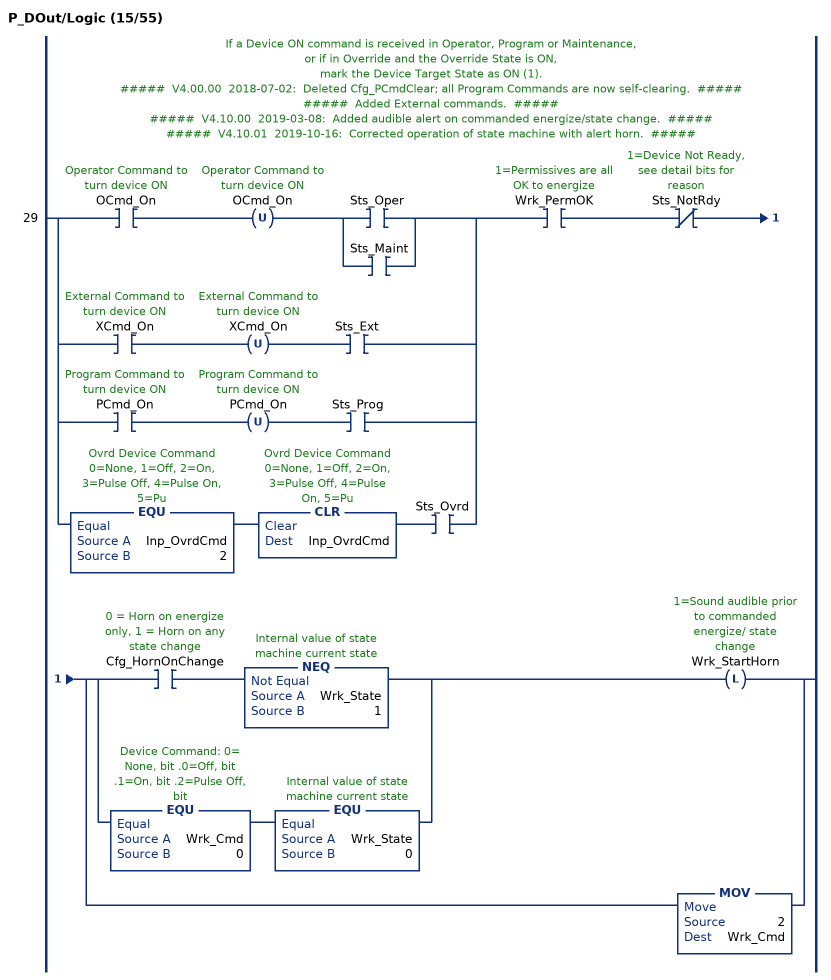
   // If a Device ON command is received in Operator, Program or Maintenance,
   // or if in Override and the Override State is ON,
   // mark the Device Target State as ON (1).
   // #####  V4.00.00  2018-07-02:  Deleted Cfg_PCmdClear; all Program Commands are now self-clearing.  #####
   // #####  Added External commands.  #####
   // #####  V4.10.00  2019-03-08:  Added audible alert on commanded energize/state change.  #####
   // #####  V4.10.01  2019-10-16:  Corrected operation of state machine with alert horn.  #####
   29: [XIC(OCmd_On) OTU(OCmd_On) [XIC(Sts_Oper) ,XIC(Sts_Maint) ] ,XIC(XCmd_On) OTU(XCmd_On) XIC(Sts_Ext) ,XIC(PCmd_On) OTU(PCmd_On) XIC(Sts_Prog) ,EQU(Inp_OvrdCmd,2) CLR(Inp_OvrdCmd) XIC(Sts_Ovrd) ]XIC(Wrk_PermOK)XIO(Sts_NotRdy)[[XIC(Cfg_HornOnChange) NEQ(Wrk_State,1) ,EQU(Wrk_Cmd,0) EQU(Wrk_State,0) ] OTL(Wrk_StartHorn) ,MOV(2,Wrk_Cmd) ];
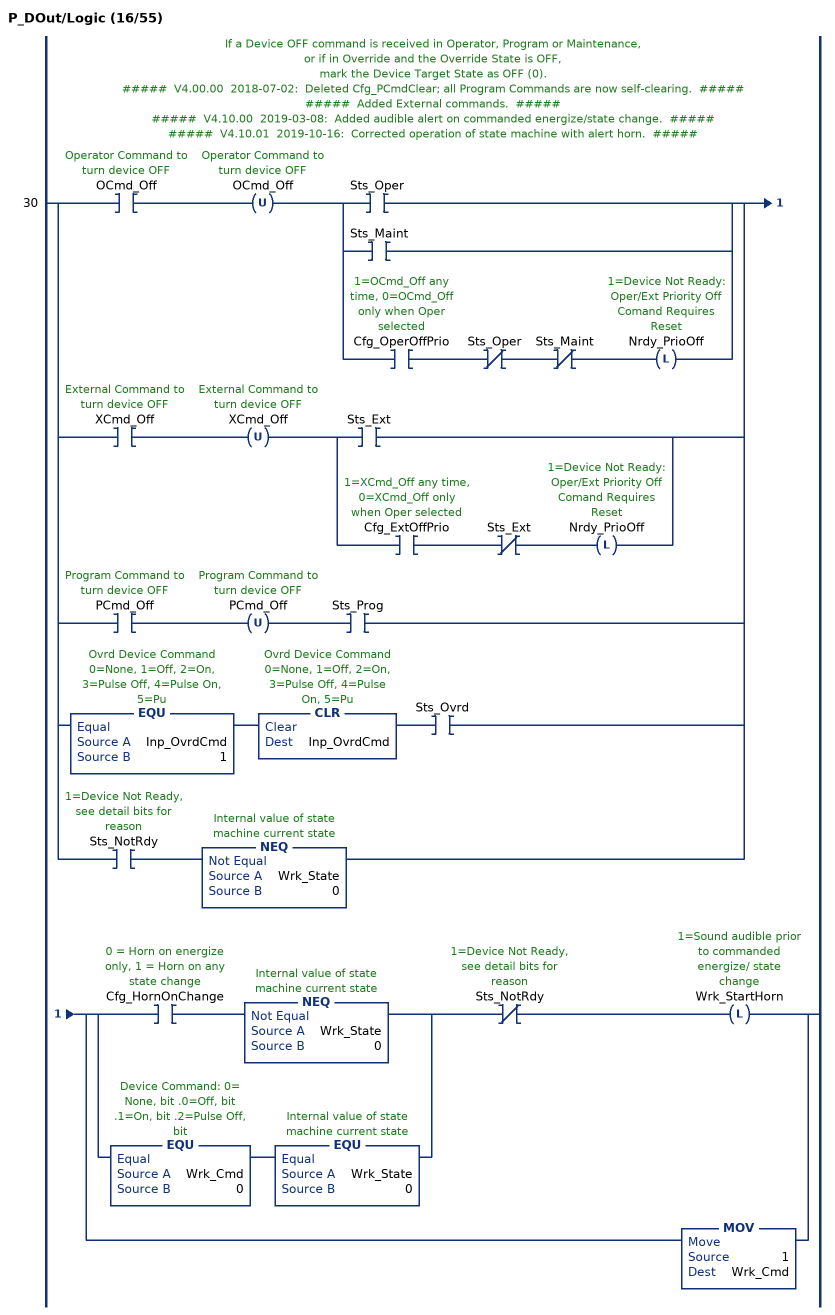
   // If a Device OFF command is received in Operator, Program or Maintenance,
   // or if in Override and the Override State is OFF,
   // mark the Device Target State as OFF (0).
   // #####  V4.00.00  2018-07-02:  Deleted Cfg_PCmdClear; all Program Commands are now self-clearing.  #####
   // #####  Added External commands.  #####
   // #####  V4.10.00  2019-03-08:  Added audible alert on commanded energize/state change.  #####
   // #####  V4.10.01  2019-10-16:  Corrected operation of state machine with alert horn.  #####
   30: [XIC(OCmd_Off) OTU(OCmd_Off) [XIC(Sts_Oper) ,XIC(Sts_Maint) ,XIC(Cfg_OperOffPrio) XIO(Sts_Oper) XIO(Sts_Maint) OTL(Nrdy_PrioOff) ] ,XIC(XCmd_Off) OTU(XCmd_Off) [XIC(Sts_Ext) ,XIC(Cfg_ExtOffPrio) XIO(Sts_Ext) OTL(Nrdy_PrioOff) ] ,XIC(PCmd_Off) OTU(PCmd_Off) XIC(Sts_Prog) ,EQU(Inp_OvrdCmd,1) CLR(Inp_OvrdCmd) XIC(Sts_Ovrd) ,XIC(Sts_NotRdy) NEQ(Wrk_State,0) ][[XIC(Cfg_HornOnChange) NEQ(Wrk_State,0) ,EQU(Wrk_Cmd,0) EQU(Wrk_State,0) ] XIO(Sts_NotRdy) OTL(Wrk_StartHorn) ,MOV(1,Wrk_Cmd) ];
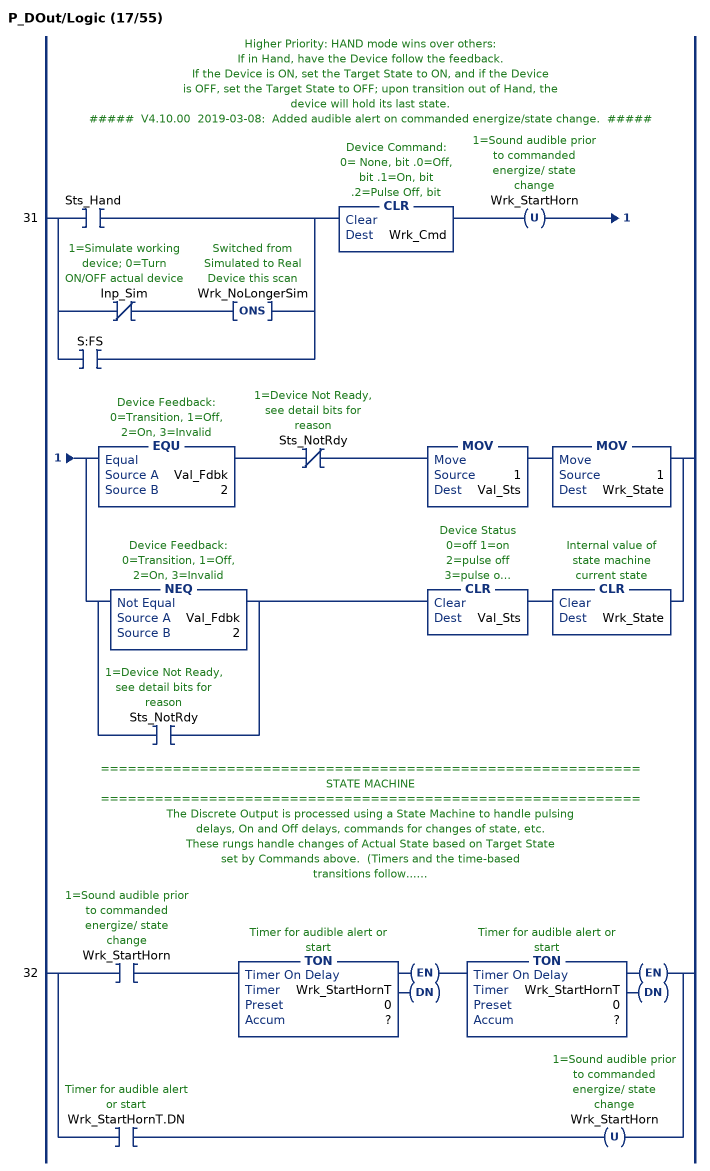
   // Higher Priority: HAND mode wins over others:
   // If in Hand, have the Device follow the feedback.
   // If the Device is ON, set the Target State to ON, and if the Device
   // is OFF, set the Target State to OFF; upon transition out of Hand, the
   // device will hold its last state.
   // #####  V4.10.00  2019-03-08:  Added audible alert on commanded energize/state change.  #####
   31: [XIC(Sts_Hand) ,XIO(Inp_Sim) ONS(Wrk_NoLongerSim) ,XIC(S:FS) ]CLR(Wrk_Cmd)OTU(Wrk_StartHorn)[EQU(Val_Fdbk,2) XIO(Sts_NotRdy) MOV(1,Val_Sts) MOV(1,Wrk_State) ,[NEQ(Val_Fdbk,2) ,XIC(Sts_NotRdy) ] CLR(Val_Sts) CLR(Wrk_State) ];
   // ============================================================
   // STATE MACHINE
   // ============================================================
   // The Discrete Output is processed using a State Machine to handle pulsing
   // delays, On and Off delays, commands for changes of state, etc.
   // These rungs handle changes of Actual State based on Target State
   // set by Commands above.  (Timers and the time-based
   // transitions follow...)
   // See the Timing Diagrams and state tables in the Reference
   // Manual for details on the state machine.
   // On Prestart Horn - Sound the horn for the configured time.
   // #####  V4.10.01  2019-10-16:  Corrected operation of state machine with alert horn.  #####
   32: [XIC(Wrk_StartHorn) TON(Wrk_StartHornT,?,?) TON(Wrk_StartHornT,?,?) ,XIC(Wrk_StartHornT.DN) OTU(Wrk_StartHorn) ];
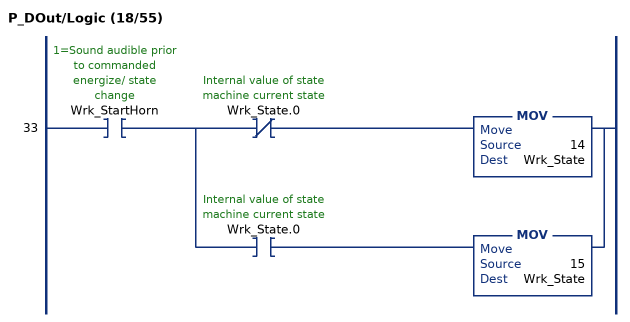
   33: XIC(Wrk_StartHorn)[XIO(Wrk_State.0) MOV(14,Wrk_State) ,XIC(Wrk_State.0) MOV(15,Wrk_State) ];
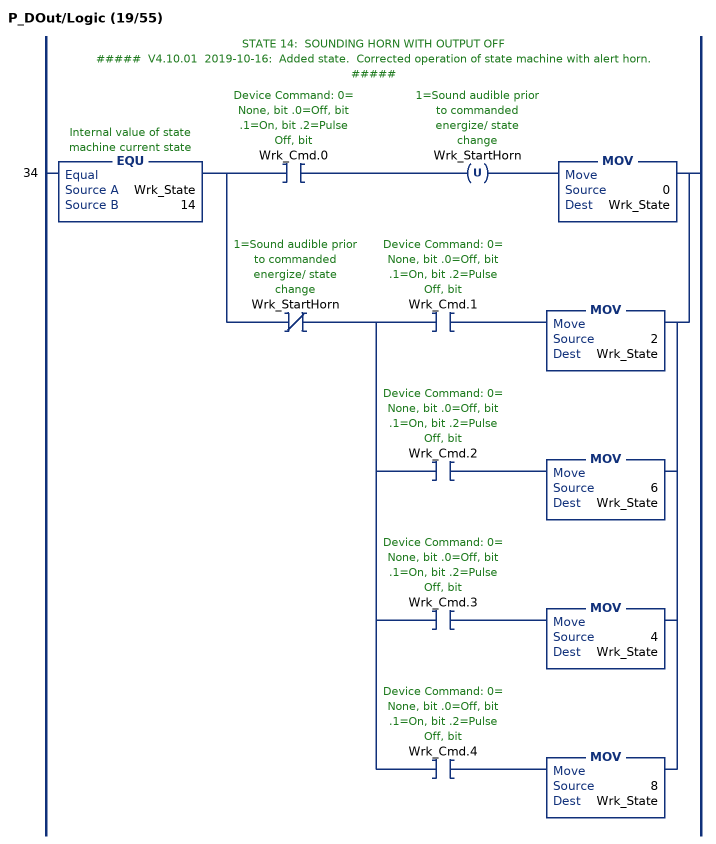
   // STATE 14:  SOUNDING HORN WITH OUTPUT OFF
   // #####  V4.10.01  2019-10-16:  Added state.  Corrected operation of state machine with alert horn.  #####
   34: EQU(Wrk_State,14)[XIC(Wrk_Cmd.0) OTU(Wrk_StartHorn) MOV(0,Wrk_State) ,XIO(Wrk_StartHorn) [XIC(Wrk_Cmd.1) MOV(2,Wrk_State) ,XIC(Wrk_Cmd.2) MOV(6,Wrk_State) ,XIC(Wrk_Cmd.3) MOV(4,Wrk_State) ,XIC(Wrk_Cmd.4) MOV(8,Wrk_State) ] ];
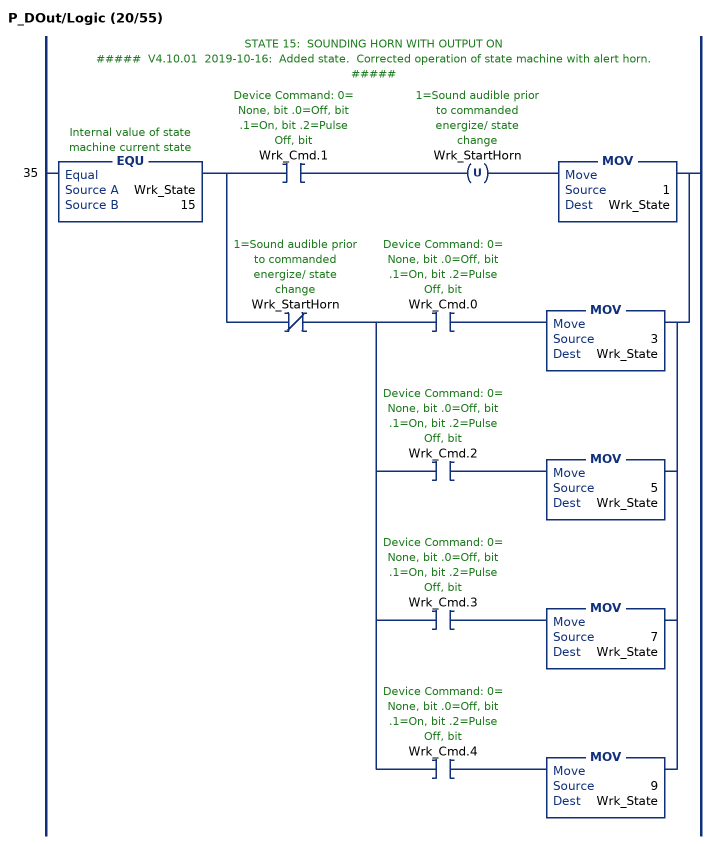
   // STATE 15:  SOUNDING HORN WITH OUTPUT ON
   // #####  V4.10.01  2019-10-16:  Added state.  Corrected operation of state machine with alert horn.  #####
   35: EQU(Wrk_State,15)[XIC(Wrk_Cmd.1) OTU(Wrk_StartHorn) MOV(1,Wrk_State) ,XIO(Wrk_StartHorn) [XIC(Wrk_Cmd.0) MOV(3,Wrk_State) ,XIC(Wrk_Cmd.2) MOV(5,Wrk_State) ,XIC(Wrk_Cmd.3) MOV(7,Wrk_State) ,XIC(Wrk_Cmd.4) MOV(9,Wrk_State) ] ];
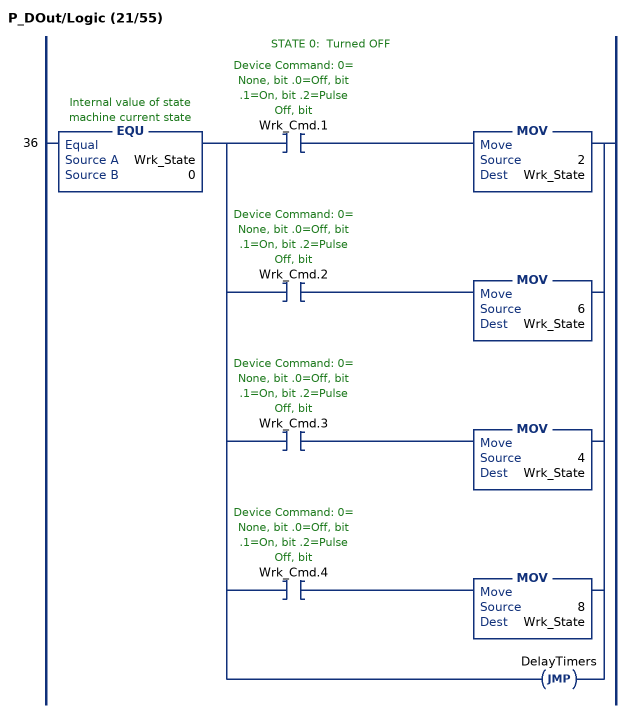
   // STATE 0:  Turned OFF
   36: EQU(Wrk_State,0)[XIC(Wrk_Cmd.1) MOV(2,Wrk_State) ,XIC(Wrk_Cmd.2) MOV(6,Wrk_State) ,XIC(Wrk_Cmd.3) MOV(4,Wrk_State) ,XIC(Wrk_Cmd.4) MOV(8,Wrk_State) ,JMP(DelayTimers) ];
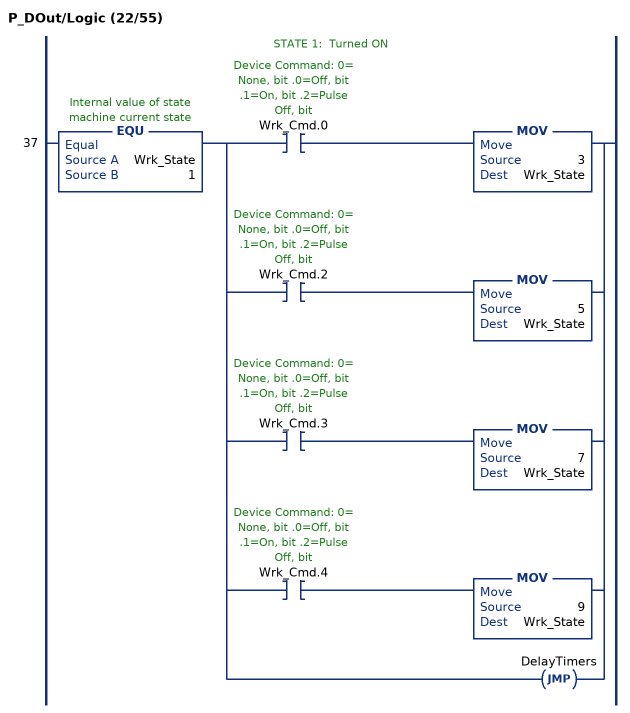
   // STATE 1:  Turned ON
   37: EQU(Wrk_State,1)[XIC(Wrk_Cmd.0) MOV(3,Wrk_State) ,XIC(Wrk_Cmd.2) MOV(5,Wrk_State) ,XIC(Wrk_Cmd.3) MOV(7,Wrk_State) ,XIC(Wrk_Cmd.4) MOV(9,Wrk_State) ,JMP(DelayTimers) ];
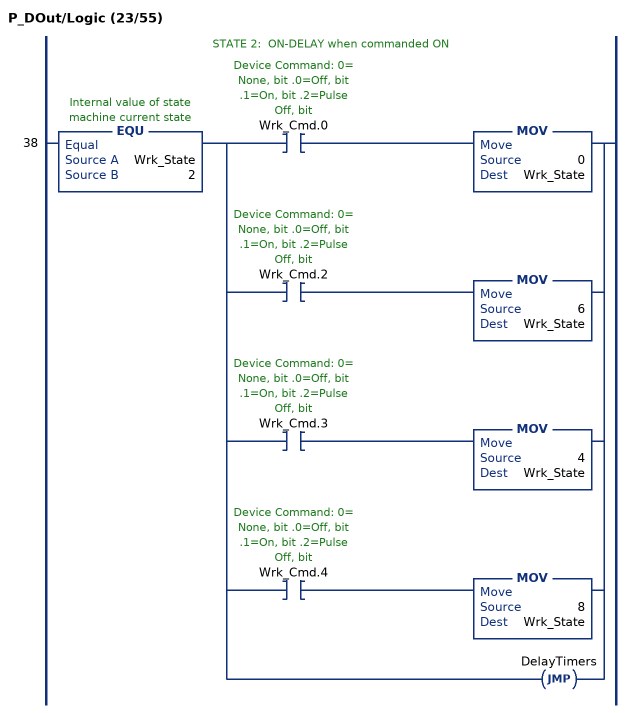
   // STATE 2:  ON-DELAY when commanded ON
   38: EQU(Wrk_State,2)[XIC(Wrk_Cmd.0) MOV(0,Wrk_State) ,XIC(Wrk_Cmd.2) MOV(6,Wrk_State) ,XIC(Wrk_Cmd.3) MOV(4,Wrk_State) ,XIC(Wrk_Cmd.4) MOV(8,Wrk_State) ,JMP(DelayTimers) ];
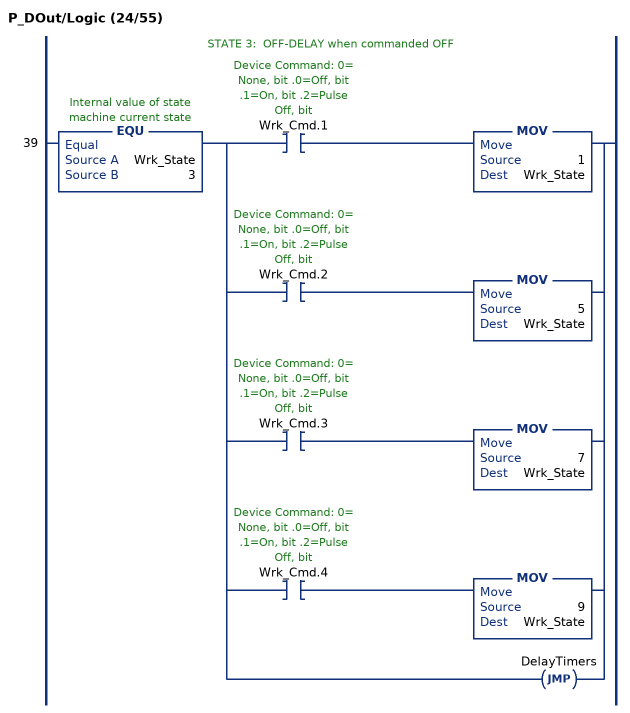
   // STATE 3:  OFF-DELAY when commanded OFF
   39: EQU(Wrk_State,3)[XIC(Wrk_Cmd.1) MOV(1,Wrk_State) ,XIC(Wrk_Cmd.2) MOV(5,Wrk_State) ,XIC(Wrk_Cmd.3) MOV(7,Wrk_State) ,XIC(Wrk_Cmd.4) MOV(9,Wrk_State) ,JMP(DelayTimers) ];
